// TIA Portal V17 export
// export: Created 2024-09-02T12:49:58.764909Z, ExportSetting WithDefaults, DisplayName Totally Integrated Automation Portal, DisplayVersion V17, DisplayName TIA Portal Openness, DisplayVersion V17, DisplayName TIA Portal Version Control Interface, DisplayVersion V17, DisplayName STEP 7 Professional, DisplayVersion V17, DisplayName STEP 7 Safety, DisplayVersion V17, DisplayName WinCC Professional, DisplayVersion V17
DATA_BLOCK "DB_Interface_HMI_Extension"   // DB12
{ S7_Optimized_Access := 'TRUE'; DB_Accessible_From_OPC_UA := 'FALSE' }
AUTHOR : SIEMENS
FAMILY : VW_ADDON
NAME : GENERAL
VERSION : 1.1
// stored: AutoNumber true, DBAccessibleFromOPCUA false, IsOnlyStoredInLoadMemory false, IsRetainMemResEnabled false, IsWriteProtectedInAS false, MemoryReserve 0
   VAR
      BildPanelControl_UhrzeitStellen : Struct   // Screen "Panel Control" Set Date and Time
         EingabeZeit : Date_And_Time := DT#18-5-1-12:0:0.000;   // Eingabe der Uhrzeit und des Datum am Panel im Bild Panel Control / Enter the time and date on the Panel in the Panel Control screen.
         UhrzeitStellen : Bool;   // Übernahme der Uhrzeit und des Datum / Acceptance of time and date
      END_STRUCT;
   END_VAR
BEGIN
END_DATA_BLOCK
